(* CoDeSys 2.3 export: PROC_ERR_SENSORS.EXP *)

(* POU 60_Error handling/Process Errors/proc_Err_Sensors, ST *)
PROGRAM proc_Err_Sensors
VAR
	ProcessErr1_fb				: handleError;

END_VAR
VAR CONSTANT

END_VAR
;
END_PROGRAM
